(* IEC 61131-3 sources: Hydro-Leak-Detection/, 3 files *)

(* ---- Hydro_Leak_Detection.st ---- *)
PROGRAM Hydro_Leak_Detection
VAR
    // --- Hardware Inputs (Mapped to Beckhoff ELM3148) ---
    iRawAnalogInput     AT %I* : INT;   // Raw 4-20mA input from DLS panel (load cell)
    bStartTestCycle             : BOOL; // Triggered by FAT rig operator to begin leak test

    // --- System Configuration Constants (1kg Top-Down Architecture) ---
    c_iRawMin           : INT  := 0;       // Raw integer value at 4mA (Beckhoff specific, often 0)
    c_iRawMax           : INT  := 32767;   // Raw integer value at 20mA (Beckhoff 16-bit)
    c_rSensorCapacity   : REAL := 1000.0;  // 1kg load cell full-scale (in grams)
    c_tSettleTime       : TIME := T#3S;    // 3-second mechanical deadband for suspension swing

    // --- Internal Logic Variables ---
    rAbsoluteMass       : REAL; // Total mass currently hanging on the sensor (grams)
    rTareMass           : REAL; // Captured weight of the empty bottle (~54g)
    bTareComplete       : BOOL; // Flag: system is zeroed and ready
    rActiveLeakMass     : REAL; // Calculated accumulated leak (grams → ml, 1g = 1ml)

    // --- Function Blocks ---
    fbSettleTimer       : TON;      // Deadband timer before tare capture
    fbTareTrigger       : R_TRIG;   // Rising edge: capture tare only once
END_VAR

// ==============================================================================
// 1. Analog Input Scaling (4-20mA → Grams)
// ==============================================================================
// Convert the raw Beckhoff integer into a percentage of full-scale, then
// multiply by the 1000g load cell capacity.
IF c_iRawMax > c_iRawMin THEN
    rAbsoluteMass := (INT_TO_REAL(iRawAnalogInput - c_iRawMin) /
                      INT_TO_REAL(c_iRawMax - c_iRawMin)) * c_rSensorCapacity;
ELSE
    rAbsoluteMass := 0.0;   // Prevent divide-by-zero on misconfigured constants
END_IF

// ==============================================================================
// 2. Mechanical Deadband & Tare Logic
// ==============================================================================
// Allow the hanging bottle to stop swinging before capturing the tare weight.
fbSettleTimer(IN := bStartTestCycle, PT := c_tSettleTime);

// Capture the tare mass exactly once when the settle timer completes.
fbTareTrigger(CLK := fbSettleTimer.Q);

IF fbTareTrigger.Q THEN
    rTareMass     := rAbsoluteMass;
    bTareComplete := TRUE;
END_IF

// Clear all state when the operator ends the test cycle.
IF NOT bStartTestCycle THEN
    bTareComplete    := FALSE;
    rTareMass        := 0.0;
    rActiveLeakMass  := 0.0;
END_IF

// ==============================================================================
// 3. Active Leak Measurement  (1g = 1ml — gravimetric equivalence for water)
// ==============================================================================
// Calculate cumulative leaked volume only after a valid tare has been taken.
IF bTareComplete THEN
    rActiveLeakMass := rAbsoluteMass - rTareMass;

    // Clamp negative readings caused by ambient vibration / sensor noise.
    IF rActiveLeakMass < 0.0 THEN
        rActiveLeakMass := 0.0;
    END_IF
ELSE
    rActiveLeakMass := 0.0;   // Output zero while the system is still settling
END_IF

// rActiveLeakMass [g] directly represents leaked volume [ml] of hydraulic fluid.
// Log or trend this variable in TwinCAT Scope / SCADA for Hydro FAT reporting.

(* ---- LVDT_Leak_Detection.st ---- *)
PROGRAM LVDT_Leak_Detection
VAR
    // --- Hardware Inputs (Mapped to Beckhoff EL3064 / ELM3104) ---
    iRawAnalogInput     AT %I* : INT;   // Raw 4-20mA input from LVDT signal conditioner
    bStartTestCycle             : BOOL; // Triggered by FAT rig operator to begin leak test

    // --- System Configuration Constants ---
    // LVDT (Linear Variable Differential Transformer) mounted vertically above
    // the leak-collection vessel. The ferromagnetic core is attached to a float
    // that rises as fluid accumulates, producing an upward displacement signal.
    c_iRawMin           : INT  := 0;       // Raw integer value at 4mA  (Beckhoff 16-bit)
    c_iRawMax           : INT  := 32767;   // Raw integer value at 20mA (Beckhoff 16-bit)
    c_rLVDTFullStroke   : REAL := 50.0;    // LVDT full mechanical stroke (mm), e.g. ±25mm = 50mm total
    c_rVesselAreaCm2    : REAL := 19.635;  // Collection vessel internal cross-section (cm²)
                                           // Example: Ø50mm circular vessel → π×(2.5)² ≈ 19.635 cm²
    c_tSettleTime       : TIME := T#3S;    // 3-second deadband: float stabilisation after placement

    // --- Internal Logic Variables ---
    rDisplacementMM     : REAL; // Scaled LVDT displacement from zero reference (mm)
    rTareDisplacement   : REAL; // Captured zero-level displacement (float at rest, empty vessel)
    bTareComplete       : BOOL; // Flag: system zeroed and ready for measurement
    rNetDisplacementMM  : REAL; // Displacement relative to tare position (mm of level rise)
    rActiveLeakVolume   : REAL; // Accumulated leak volume in millilitres

    // --- Function Blocks ---
    fbSettleTimer       : TON;      // Deadband timer — wait for float to stabilise
    fbTareTrigger       : R_TRIG;   // Rising edge: capture tare zero once
END_VAR

// ==============================================================================
// 1. Analog Input Scaling (4-20mA → Displacement in mm)
// ==============================================================================
// The LVDT conditioner outputs 4mA at minimum core displacement (float at
// bottom / vessel empty) and 20mA at maximum upward displacement (vessel full).
// Scale the raw Beckhoff integer to a physical displacement in millimetres.
IF c_iRawMax > c_iRawMin THEN
    rDisplacementMM := (INT_TO_REAL(iRawAnalogInput - c_iRawMin) /
                        INT_TO_REAL(c_iRawMax - c_iRawMin)) * c_rLVDTFullStroke;
ELSE
    rDisplacementMM := 0.0;   // Prevent divide-by-zero on misconfigured constants
END_IF

// ==============================================================================
// 2. Float Stabilisation & Tare Logic
// ==============================================================================
// Wait for the collection vessel float to settle before capturing the zero
// reference.  Any residual fluid from a previous test causes a non-zero tare
// which is correctly zeroed out by this logic.
fbSettleTimer(IN := bStartTestCycle, PT := c_tSettleTime);

fbTareTrigger(CLK := fbSettleTimer.Q);

IF fbTareTrigger.Q THEN
    rTareDisplacement := rDisplacementMM;
    bTareComplete     := TRUE;
END_IF

// Clear all state when the operator ends the test cycle.
IF NOT bStartTestCycle THEN
    bTareComplete      := FALSE;
    rTareDisplacement  := 0.0;
    rNetDisplacementMM := 0.0;
    rActiveLeakVolume  := 0.0;
END_IF

// ==============================================================================
// 3. Active Leak Measurement  (displacement → volume)
// ==============================================================================
// Volume (ml) = cross-sectional area (cm²) × level rise (cm)
//             = c_rVesselAreaCm2 × (rNetDisplacementMM / 10.0)
//
// Unit chain:  [cm²] × [mm / 10  = cm]  →  [cm³]  ≡  [ml]
IF bTareComplete THEN
    rNetDisplacementMM := rDisplacementMM - rTareDisplacement;

    // Clamp negative values: LVDT noise or minor float oscillation
    IF rNetDisplacementMM < 0.0 THEN
        rNetDisplacementMM := 0.0;
    END_IF

    rActiveLeakVolume := c_rVesselAreaCm2 * (rNetDisplacementMM / 10.0);
ELSE
    rNetDisplacementMM := 0.0;
    rActiveLeakVolume  := 0.0;   // Output zero while the system is still settling
END_IF

// rActiveLeakVolume [ml] represents the total accumulated hydraulic fluid leak.
// rNetDisplacementMM [mm] is available as a raw diagnostic / calibration signal.
// Log or trend these variables in TwinCAT Scope / SCADA for Hydro FAT reporting.

(* ---- Ultrasonic_Leak_Detection.st ---- *)
PROGRAM Ultrasonic_Leak_Detection
VAR
    // --- Hardware Inputs (Mapped to Beckhoff EL3064 / ELM3104) ---
    iRawAnalogInput     AT %I* : INT;   // Raw 4-20mA input from ultrasonic level transmitter
    bStartTestCycle             : BOOL; // Triggered by FAT rig operator to begin leak test

    // --- System Configuration Constants ---
    // Non-contact ultrasonic level transmitter mounted above the open-top
    // leak-collection vessel, facing downward.  The transmitter emits ultrasonic
    // pulses; time-of-flight to the fluid surface is converted to a 4-20mA signal.
    //
    // Wiring convention used here (verify against specific transmitter datasheet):
    //   4mA  → empty vessel  (maximum distance from sensor to vessel floor)
    //   20mA → full vessel   (minimum distance, fluid surface near sensor)
    // This gives a DIRECT relationship: higher current = higher fluid level.
    c_iRawMin           : INT  := 0;       // Raw integer at 4mA  (Beckhoff 16-bit)
    c_iRawMax           : INT  := 32767;   // Raw integer at 20mA (Beckhoff 16-bit)
    c_rSensorRangeMM    : REAL := 300.0;   // Transmitter measurement span (mm), e.g. 0–300mm level
    c_rVesselAreaCm2    : REAL := 19.635;  // Collection vessel internal cross-section (cm²)
                                           // Example: Ø50mm circular vessel → π×(2.5)² ≈ 19.635 cm²
    c_tSettleTime       : TIME := T#3S;    // 3-second deadband: allow ultrasonic reading to stabilise
    c_rNoiseThreshMM    : REAL := 0.5;     // Dead-band below which level change is treated as noise (mm)

    // --- Internal Logic Variables ---
    rLevelMM            : REAL; // Scaled fluid level in the collection vessel (mm)
    rTareLevel          : REAL; // Captured zero-level at start of test (residual fluid baseline)
    bTareComplete       : BOOL; // Flag: system zeroed and ready
    rNetLevelMM         : REAL; // Level rise relative to tare (mm)
    rActiveLeakVolume   : REAL; // Accumulated leak volume (ml)

    // --- Function Blocks ---
    fbSettleTimer       : TON;      // Deadband timer — wait for ultrasonic echo to stabilise
    fbTareTrigger       : R_TRIG;   // Rising edge: capture tare zero once
END_VAR

// ==============================================================================
// 1. Analog Input Scaling (4-20mA → Fluid Level in mm)
// ==============================================================================
// Scale the Beckhoff raw integer to a physical fluid-level reading in mm.
// At 4mA the vessel is empty (level = 0mm); at 20mA level = c_rSensorRangeMM.
IF c_iRawMax > c_iRawMin THEN
    rLevelMM := (INT_TO_REAL(iRawAnalogInput - c_iRawMin) /
                 INT_TO_REAL(c_iRawMax - c_iRawMin)) * c_rSensorRangeMM;
ELSE
    rLevelMM := 0.0;   // Prevent divide-by-zero on misconfigured constants
END_IF

// ==============================================================================
// 2. Echo Stabilisation & Tare Logic
// ==============================================================================
// Ultrasonic readings can be momentarily disturbed by vibration, turbulence, or
// foam on the fluid surface.  The settle timer allows the echo to stabilise
// before the zero-reference (tare) is captured.
fbSettleTimer(IN := bStartTestCycle, PT := c_tSettleTime);

fbTareTrigger(CLK := fbSettleTimer.Q);

IF fbTareTrigger.Q THEN
    rTareLevel    := rLevelMM;
    bTareComplete := TRUE;
END_IF

// Clear all state when the operator ends the test cycle.
IF NOT bStartTestCycle THEN
    bTareComplete     := FALSE;
    rTareLevel        := 0.0;
    rNetLevelMM       := 0.0;
    rActiveLeakVolume := 0.0;
END_IF

// ==============================================================================
// 3. Active Leak Measurement  (level rise → volume)
// ==============================================================================
// Volume (ml) = cross-sectional area (cm²) × level rise (cm)
//             = c_rVesselAreaCm2 × (rNetLevelMM / 10.0)
//
// Unit chain:  [cm²] × [mm / 10 = cm]  →  [cm³]  ≡  [ml]
IF bTareComplete THEN
    rNetLevelMM := rLevelMM - rTareLevel;

    // Apply noise dead-band: ignore sub-threshold level fluctuations
    IF rNetLevelMM < c_rNoiseThreshMM THEN
        rNetLevelMM := 0.0;
    END_IF

    rActiveLeakVolume := c_rVesselAreaCm2 * (rNetLevelMM / 10.0);
ELSE
    rNetLevelMM       := 0.0;
    rActiveLeakVolume := 0.0;   // Output zero while the system is still settling
END_IF

// rActiveLeakVolume [ml] represents the total accumulated hydraulic fluid leak.
// rNetLevelMM [mm] is available as a raw diagnostic / calibration signal.
//
// NOTE — Foam / Turbulence mitigation: for highly turbulent leaks consider
// enabling the transmitter's internal averaging filter (if available) and
// increasing c_tSettleTime to T#5S.  Alternatively, a first-order IIR software
// filter can be applied to rLevelMM before the tare/net calculation.
//
// Log or trend rActiveLeakVolume in TwinCAT Scope / SCADA for Hydro FAT reporting.
